SUBAPPLICATION GreenWhiteBackground_Knickdeichsel_senken (* Subapplication Type *)
  (* Standard: 61499-2 *)
  (* Version 1.0, 2023-02-11, franz *)
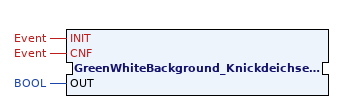
  EVENT_INPUT
    INIT;
    CNF;
  END_EVENT
  VAR_INPUT
    OUT : BOOL;
  END_VAR
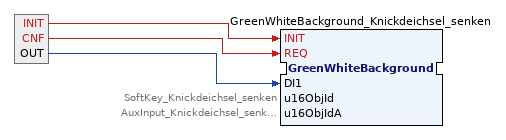
  SUBAPPS
    GreenWhiteBackground_Knickdeichsel_senken : GreenWhiteBackground(u16ObjId := SoftKey_Knickdeichsel_senken, u16ObjIdA := AuxInput_Knickdeichsel_senken);
  END_SUBAPPS
  EVENT_CONNECTIONS
    INIT TO GreenWhiteBackground_Knickdeichsel_senken.INIT;
    CNF TO GreenWhiteBackground_Knickdeichsel_senken.REQ;
  END_CONNECTIONS
  DATA_CONNECTIONS
    OUT TO GreenWhiteBackground_Knickdeichsel_senken.DI1;
  END_CONNECTIONS
END_SUBAPPLICATION
